// TIA Portal V16 export
// export: Created 2023-06-21T17:06:27.0231194Z, ExportSetting WithDefaults, DisplayName Totally Integrated Automation Portal, DisplayVersion V16 Update 4, DisplayName TIA Portal Version Control Interface, DisplayVersion V16 Update 2, DisplayName TIA Portal Openness, DisplayVersion V16 Update 4, DisplayName SINAMICS Startdrive Advanced, DisplayVersion V16, DisplayName SINAMICS Startdrive G130, G150, S120, S150, SINAMICS MV, S210, DisplayVersion V16, DisplayName SINAMICS Startdrive G110M, G120, G120C, G120D, G120P, DisplayVersion V16, DisplayName STEP 7 Professional, DisplayVersion V16 Update 4, DisplayName STEP 7 Safety, DisplayVersion V16, DisplayName Soft Starter ES, DisplayVersion V16, DisplayName WinCC Advanced, DisplayVersion V16 Update 4
FUNCTION "Data_Treatment" : Void   // FC2, LAD
{ S7_Optimized_Access := 'TRUE' }
VERSION : 0.1
// stored: AutoNumber true, IsIECCheckEnabled false, SetENOAutomatically false, UDAEnableTagReadback false
BEGIN

REGION Network 1: Extrusora 1
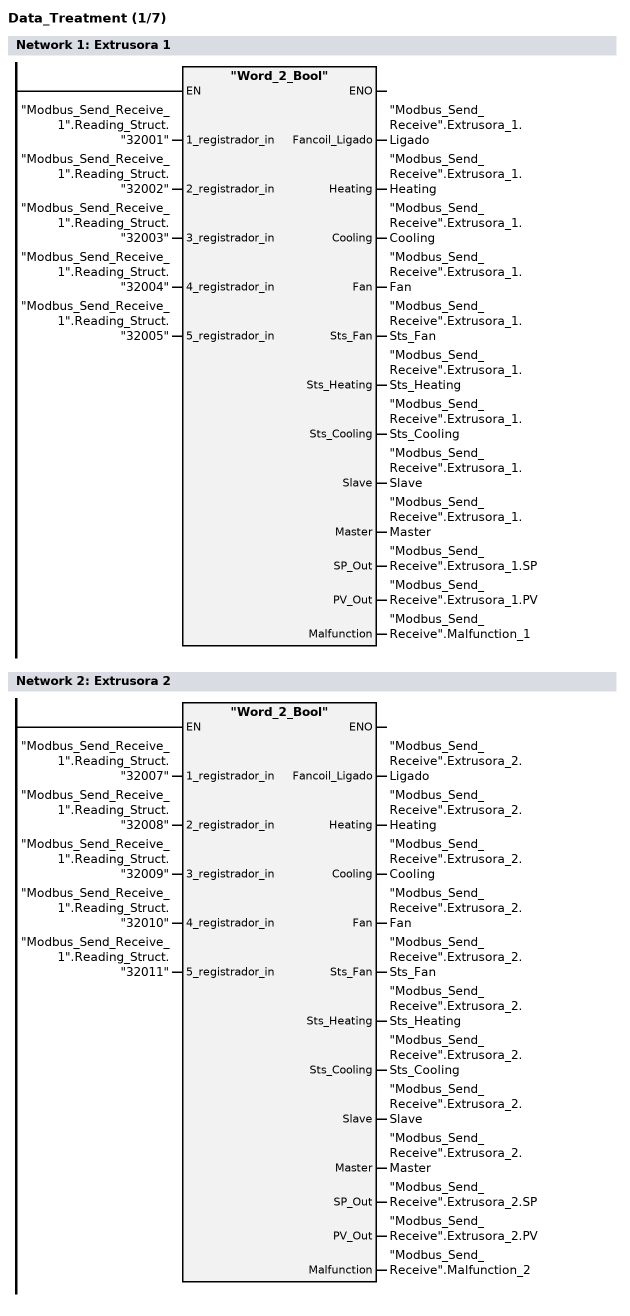
   RUNG wire#powerrail
      "Word_2_Bool"("1_registrador_in" := "Modbus_Send_Receive_1".Reading_Struct."32001", "2_registrador_in" := "Modbus_Send_Receive_1".Reading_Struct."32002", "3_registrador_in" := "Modbus_Send_Receive_1".Reading_Struct."32003", "4_registrador_in" := "Modbus_Send_Receive_1".Reading_Struct."32004", "5_registrador_in" := "Modbus_Send_Receive_1".Reading_Struct."32005", Fancoil_Ligado => "Modbus_Send_Receive".Extrusora_1.Ligado, Heating => "Modbus_Send_Receive".Extrusora_1.Heating, Cooling => "Modbus_Send_Receive".Extrusora_1.Cooling, Fan => "Modbus_Send_Receive".Extrusora_1.Fan, Sts_Fan => "Modbus_Send_Receive".Extrusora_1.Sts_Fan, Sts_Heating => "Modbus_Send_Receive".Extrusora_1.Sts_Heating, Sts_Cooling => "Modbus_Send_Receive".Extrusora_1.Sts_Cooling, Slave => "Modbus_Send_Receive".Extrusora_1.Slave, Master => "Modbus_Send_Receive".Extrusora_1.Master, SP_Out => "Modbus_Send_Receive".Extrusora_1.SP, PV_Out => "Modbus_Send_Receive".Extrusora_1.PV, Malfunction => "Modbus_Send_Receive".Malfunction_1)
   END_RUNG
   // the same network as SCL:
   "Word_2_Bool"("1_registrador_in" := "Modbus_Send_Receive_1".Reading_Struct."32001",
                 "2_registrador_in" := "Modbus_Send_Receive_1".Reading_Struct."32002",
                 "3_registrador_in" := "Modbus_Send_Receive_1".Reading_Struct."32003",
                 "4_registrador_in" := "Modbus_Send_Receive_1".Reading_Struct."32004",
                 "5_registrador_in" := "Modbus_Send_Receive_1".Reading_Struct."32005",
                 Fancoil_Ligado => "Modbus_Send_Receive".Extrusora_1.Ligado,
                 Heating => "Modbus_Send_Receive".Extrusora_1.Heating,
                 Cooling => "Modbus_Send_Receive".Extrusora_1.Cooling,
                 Fan => "Modbus_Send_Receive".Extrusora_1.Fan,
                 Sts_Fan => "Modbus_Send_Receive".Extrusora_1.Sts_Fan,
                 Sts_Heating => "Modbus_Send_Receive".Extrusora_1.Sts_Heating,
                 Sts_Cooling => "Modbus_Send_Receive".Extrusora_1.Sts_Cooling,
                 Slave => "Modbus_Send_Receive".Extrusora_1.Slave,
                 Master => "Modbus_Send_Receive".Extrusora_1.Master,
                 SP_Out => "Modbus_Send_Receive".Extrusora_1.SP,
                 PV_Out => "Modbus_Send_Receive".Extrusora_1.PV,
                 Malfunction => "Modbus_Send_Receive".Malfunction_1);
END_REGION

REGION Network 2: Extrusora 2
   RUNG wire#powerrail
      "Word_2_Bool"("1_registrador_in" := "Modbus_Send_Receive_1".Reading_Struct."32007", "2_registrador_in" := "Modbus_Send_Receive_1".Reading_Struct."32008", "3_registrador_in" := "Modbus_Send_Receive_1".Reading_Struct."32009", "4_registrador_in" := "Modbus_Send_Receive_1".Reading_Struct."32010", "5_registrador_in" := "Modbus_Send_Receive_1".Reading_Struct."32011", Fancoil_Ligado => "Modbus_Send_Receive".Extrusora_2.Ligado, Heating => "Modbus_Send_Receive".Extrusora_2.Heating, Cooling => "Modbus_Send_Receive".Extrusora_2.Cooling, Fan => "Modbus_Send_Receive".Extrusora_2.Fan, Sts_Fan => "Modbus_Send_Receive".Extrusora_2.Sts_Fan, Sts_Heating => "Modbus_Send_Receive".Extrusora_2.Sts_Heating, Sts_Cooling => "Modbus_Send_Receive".Extrusora_2.Sts_Cooling, Slave => "Modbus_Send_Receive".Extrusora_2.Slave, Master => "Modbus_Send_Receive".Extrusora_2.Master, SP_Out => "Modbus_Send_Receive".Extrusora_2.SP, PV_Out => "Modbus_Send_Receive".Extrusora_2.PV, Malfunction => "Modbus_Send_Receive".Malfunction_2)
   END_RUNG
   // the same network as SCL:
   "Word_2_Bool"("1_registrador_in" := "Modbus_Send_Receive_1".Reading_Struct."32007",
                 "2_registrador_in" := "Modbus_Send_Receive_1".Reading_Struct."32008",
                 "3_registrador_in" := "Modbus_Send_Receive_1".Reading_Struct."32009",
                 "4_registrador_in" := "Modbus_Send_Receive_1".Reading_Struct."32010",
                 "5_registrador_in" := "Modbus_Send_Receive_1".Reading_Struct."32011",
                 Fancoil_Ligado => "Modbus_Send_Receive".Extrusora_2.Ligado,
                 Heating => "Modbus_Send_Receive".Extrusora_2.Heating,
                 Cooling => "Modbus_Send_Receive".Extrusora_2.Cooling,
                 Fan => "Modbus_Send_Receive".Extrusora_2.Fan,
                 Sts_Fan => "Modbus_Send_Receive".Extrusora_2.Sts_Fan,
                 Sts_Heating => "Modbus_Send_Receive".Extrusora_2.Sts_Heating,
                 Sts_Cooling => "Modbus_Send_Receive".Extrusora_2.Sts_Cooling,
                 Slave => "Modbus_Send_Receive".Extrusora_2.Slave,
                 Master => "Modbus_Send_Receive".Extrusora_2.Master,
                 SP_Out => "Modbus_Send_Receive".Extrusora_2.SP,
                 PV_Out => "Modbus_Send_Receive".Extrusora_2.PV,
                 Malfunction => "Modbus_Send_Receive".Malfunction_2);
END_REGION

REGION Network 3: Extrusora 3
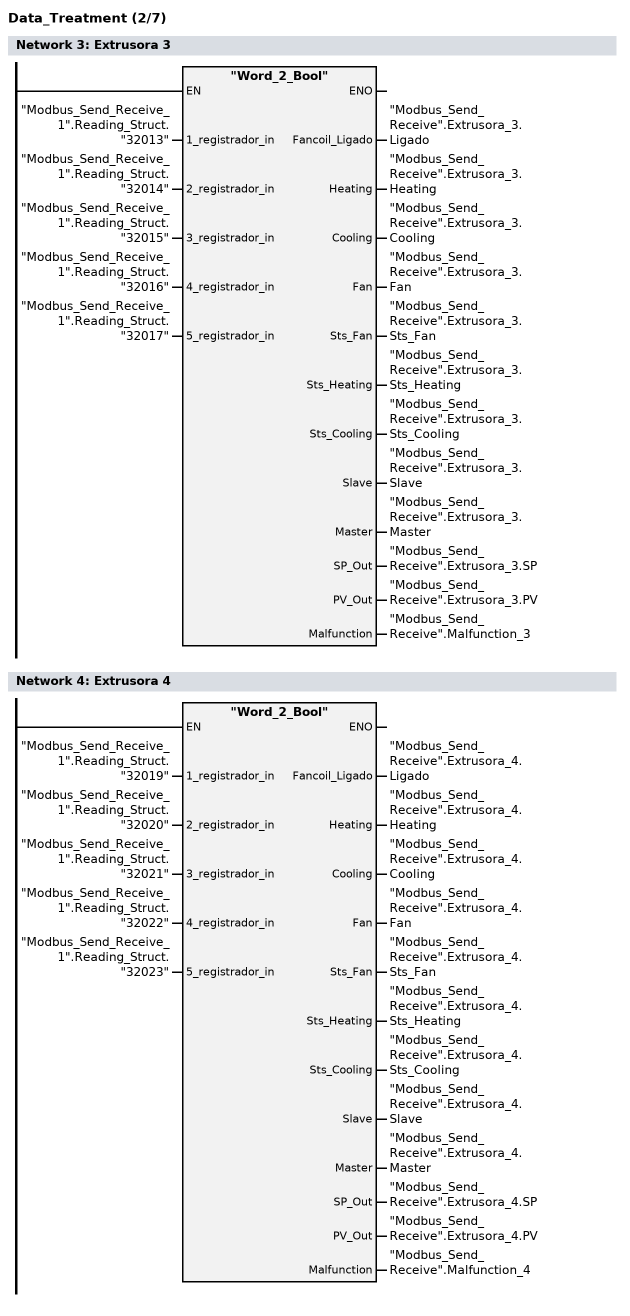
   RUNG wire#powerrail
      "Word_2_Bool"("1_registrador_in" := "Modbus_Send_Receive_1".Reading_Struct."32013", "2_registrador_in" := "Modbus_Send_Receive_1".Reading_Struct."32014", "3_registrador_in" := "Modbus_Send_Receive_1".Reading_Struct."32015", "4_registrador_in" := "Modbus_Send_Receive_1".Reading_Struct."32016", "5_registrador_in" := "Modbus_Send_Receive_1".Reading_Struct."32017", Fancoil_Ligado => "Modbus_Send_Receive".Extrusora_3.Ligado, Heating => "Modbus_Send_Receive".Extrusora_3.Heating, Cooling => "Modbus_Send_Receive".Extrusora_3.Cooling, Fan => "Modbus_Send_Receive".Extrusora_3.Fan, Sts_Fan => "Modbus_Send_Receive".Extrusora_3.Sts_Fan, Sts_Heating => "Modbus_Send_Receive".Extrusora_3.Sts_Heating, Sts_Cooling => "Modbus_Send_Receive".Extrusora_3.Sts_Cooling, Slave => "Modbus_Send_Receive".Extrusora_3.Slave, Master => "Modbus_Send_Receive".Extrusora_3.Master, SP_Out => "Modbus_Send_Receive".Extrusora_3.SP, PV_Out => "Modbus_Send_Receive".Extrusora_3.PV, Malfunction => "Modbus_Send_Receive".Malfunction_3)
   END_RUNG
   // the same network as SCL:
   "Word_2_Bool"("1_registrador_in" := "Modbus_Send_Receive_1".Reading_Struct."32013",
                 "2_registrador_in" := "Modbus_Send_Receive_1".Reading_Struct."32014",
                 "3_registrador_in" := "Modbus_Send_Receive_1".Reading_Struct."32015",
                 "4_registrador_in" := "Modbus_Send_Receive_1".Reading_Struct."32016",
                 "5_registrador_in" := "Modbus_Send_Receive_1".Reading_Struct."32017",
                 Fancoil_Ligado => "Modbus_Send_Receive".Extrusora_3.Ligado,
                 Heating => "Modbus_Send_Receive".Extrusora_3.Heating,
                 Cooling => "Modbus_Send_Receive".Extrusora_3.Cooling,
                 Fan => "Modbus_Send_Receive".Extrusora_3.Fan,
                 Sts_Fan => "Modbus_Send_Receive".Extrusora_3.Sts_Fan,
                 Sts_Heating => "Modbus_Send_Receive".Extrusora_3.Sts_Heating,
                 Sts_Cooling => "Modbus_Send_Receive".Extrusora_3.Sts_Cooling,
                 Slave => "Modbus_Send_Receive".Extrusora_3.Slave,
                 Master => "Modbus_Send_Receive".Extrusora_3.Master,
                 SP_Out => "Modbus_Send_Receive".Extrusora_3.SP,
                 PV_Out => "Modbus_Send_Receive".Extrusora_3.PV,
                 Malfunction => "Modbus_Send_Receive".Malfunction_3);
END_REGION

REGION Network 4: Extrusora 4
   RUNG wire#powerrail
      "Word_2_Bool"("1_registrador_in" := "Modbus_Send_Receive_1".Reading_Struct."32019", "2_registrador_in" := "Modbus_Send_Receive_1".Reading_Struct."32020", "3_registrador_in" := "Modbus_Send_Receive_1".Reading_Struct."32021", "4_registrador_in" := "Modbus_Send_Receive_1".Reading_Struct."32022", "5_registrador_in" := "Modbus_Send_Receive_1".Reading_Struct."32023", Fancoil_Ligado => "Modbus_Send_Receive".Extrusora_4.Ligado, Heating => "Modbus_Send_Receive".Extrusora_4.Heating, Cooling => "Modbus_Send_Receive".Extrusora_4.Cooling, Fan => "Modbus_Send_Receive".Extrusora_4.Fan, Sts_Fan => "Modbus_Send_Receive".Extrusora_4.Sts_Fan, Sts_Heating => "Modbus_Send_Receive".Extrusora_4.Sts_Heating, Sts_Cooling => "Modbus_Send_Receive".Extrusora_4.Sts_Cooling, Slave => "Modbus_Send_Receive".Extrusora_4.Slave, Master => "Modbus_Send_Receive".Extrusora_4.Master, SP_Out => "Modbus_Send_Receive".Extrusora_4.SP, PV_Out => "Modbus_Send_Receive".Extrusora_4.PV, Malfunction => "Modbus_Send_Receive".Malfunction_4)
   END_RUNG
   // the same network as SCL:
   "Word_2_Bool"("1_registrador_in" := "Modbus_Send_Receive_1".Reading_Struct."32019",
                 "2_registrador_in" := "Modbus_Send_Receive_1".Reading_Struct."32020",
                 "3_registrador_in" := "Modbus_Send_Receive_1".Reading_Struct."32021",
                 "4_registrador_in" := "Modbus_Send_Receive_1".Reading_Struct."32022",
                 "5_registrador_in" := "Modbus_Send_Receive_1".Reading_Struct."32023",
                 Fancoil_Ligado => "Modbus_Send_Receive".Extrusora_4.Ligado,
                 Heating => "Modbus_Send_Receive".Extrusora_4.Heating,
                 Cooling => "Modbus_Send_Receive".Extrusora_4.Cooling,
                 Fan => "Modbus_Send_Receive".Extrusora_4.Fan,
                 Sts_Fan => "Modbus_Send_Receive".Extrusora_4.Sts_Fan,
                 Sts_Heating => "Modbus_Send_Receive".Extrusora_4.Sts_Heating,
                 Sts_Cooling => "Modbus_Send_Receive".Extrusora_4.Sts_Cooling,
                 Slave => "Modbus_Send_Receive".Extrusora_4.Slave,
                 Master => "Modbus_Send_Receive".Extrusora_4.Master,
                 SP_Out => "Modbus_Send_Receive".Extrusora_4.SP,
                 PV_Out => "Modbus_Send_Receive".Extrusora_4.PV,
                 Malfunction => "Modbus_Send_Receive".Malfunction_4);
END_REGION

REGION Network 5: Extrusora 5
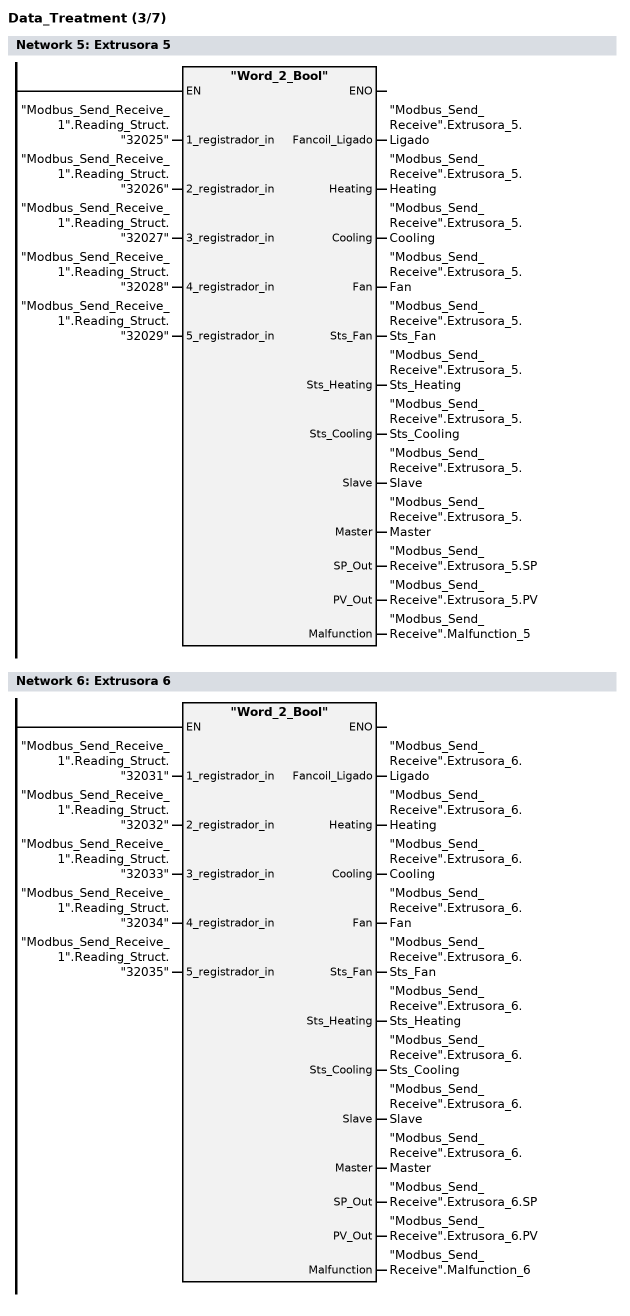
   RUNG wire#powerrail
      "Word_2_Bool"("1_registrador_in" := "Modbus_Send_Receive_1".Reading_Struct."32025", "2_registrador_in" := "Modbus_Send_Receive_1".Reading_Struct."32026", "3_registrador_in" := "Modbus_Send_Receive_1".Reading_Struct."32027", "4_registrador_in" := "Modbus_Send_Receive_1".Reading_Struct."32028", "5_registrador_in" := "Modbus_Send_Receive_1".Reading_Struct."32029", Fancoil_Ligado => "Modbus_Send_Receive".Extrusora_5.Ligado, Heating => "Modbus_Send_Receive".Extrusora_5.Heating, Cooling => "Modbus_Send_Receive".Extrusora_5.Cooling, Fan => "Modbus_Send_Receive".Extrusora_5.Fan, Sts_Fan => "Modbus_Send_Receive".Extrusora_5.Sts_Fan, Sts_Heating => "Modbus_Send_Receive".Extrusora_5.Sts_Heating, Sts_Cooling => "Modbus_Send_Receive".Extrusora_5.Sts_Cooling, Slave => "Modbus_Send_Receive".Extrusora_5.Slave, Master => "Modbus_Send_Receive".Extrusora_5.Master, SP_Out => "Modbus_Send_Receive".Extrusora_5.SP, PV_Out => "Modbus_Send_Receive".Extrusora_5.PV, Malfunction => "Modbus_Send_Receive".Malfunction_5)
   END_RUNG
   // the same network as SCL:
   "Word_2_Bool"("1_registrador_in" := "Modbus_Send_Receive_1".Reading_Struct."32025",
                 "2_registrador_in" := "Modbus_Send_Receive_1".Reading_Struct."32026",
                 "3_registrador_in" := "Modbus_Send_Receive_1".Reading_Struct."32027",
                 "4_registrador_in" := "Modbus_Send_Receive_1".Reading_Struct."32028",
                 "5_registrador_in" := "Modbus_Send_Receive_1".Reading_Struct."32029",
                 Fancoil_Ligado => "Modbus_Send_Receive".Extrusora_5.Ligado,
                 Heating => "Modbus_Send_Receive".Extrusora_5.Heating,
                 Cooling => "Modbus_Send_Receive".Extrusora_5.Cooling,
                 Fan => "Modbus_Send_Receive".Extrusora_5.Fan,
                 Sts_Fan => "Modbus_Send_Receive".Extrusora_5.Sts_Fan,
                 Sts_Heating => "Modbus_Send_Receive".Extrusora_5.Sts_Heating,
                 Sts_Cooling => "Modbus_Send_Receive".Extrusora_5.Sts_Cooling,
                 Slave => "Modbus_Send_Receive".Extrusora_5.Slave,
                 Master => "Modbus_Send_Receive".Extrusora_5.Master,
                 SP_Out => "Modbus_Send_Receive".Extrusora_5.SP,
                 PV_Out => "Modbus_Send_Receive".Extrusora_5.PV,
                 Malfunction => "Modbus_Send_Receive".Malfunction_5);
END_REGION

REGION Network 6: Extrusora 6
   RUNG wire#powerrail
      "Word_2_Bool"("1_registrador_in" := "Modbus_Send_Receive_1".Reading_Struct."32031", "2_registrador_in" := "Modbus_Send_Receive_1".Reading_Struct."32032", "3_registrador_in" := "Modbus_Send_Receive_1".Reading_Struct."32033", "4_registrador_in" := "Modbus_Send_Receive_1".Reading_Struct."32034", "5_registrador_in" := "Modbus_Send_Receive_1".Reading_Struct."32035", Fancoil_Ligado => "Modbus_Send_Receive".Extrusora_6.Ligado, Heating => "Modbus_Send_Receive".Extrusora_6.Heating, Cooling => "Modbus_Send_Receive".Extrusora_6.Cooling, Fan => "Modbus_Send_Receive".Extrusora_6.Fan, Sts_Fan => "Modbus_Send_Receive".Extrusora_6.Sts_Fan, Sts_Heating => "Modbus_Send_Receive".Extrusora_6.Sts_Heating, Sts_Cooling => "Modbus_Send_Receive".Extrusora_6.Sts_Cooling, Slave => "Modbus_Send_Receive".Extrusora_6.Slave, Master => "Modbus_Send_Receive".Extrusora_6.Master, SP_Out => "Modbus_Send_Receive".Extrusora_6.SP, PV_Out => "Modbus_Send_Receive".Extrusora_6.PV, Malfunction => "Modbus_Send_Receive".Malfunction_6)
   END_RUNG
   // the same network as SCL:
   "Word_2_Bool"("1_registrador_in" := "Modbus_Send_Receive_1".Reading_Struct."32031",
                 "2_registrador_in" := "Modbus_Send_Receive_1".Reading_Struct."32032",
                 "3_registrador_in" := "Modbus_Send_Receive_1".Reading_Struct."32033",
                 "4_registrador_in" := "Modbus_Send_Receive_1".Reading_Struct."32034",
                 "5_registrador_in" := "Modbus_Send_Receive_1".Reading_Struct."32035",
                 Fancoil_Ligado => "Modbus_Send_Receive".Extrusora_6.Ligado,
                 Heating => "Modbus_Send_Receive".Extrusora_6.Heating,
                 Cooling => "Modbus_Send_Receive".Extrusora_6.Cooling,
                 Fan => "Modbus_Send_Receive".Extrusora_6.Fan,
                 Sts_Fan => "Modbus_Send_Receive".Extrusora_6.Sts_Fan,
                 Sts_Heating => "Modbus_Send_Receive".Extrusora_6.Sts_Heating,
                 Sts_Cooling => "Modbus_Send_Receive".Extrusora_6.Sts_Cooling,
                 Slave => "Modbus_Send_Receive".Extrusora_6.Slave,
                 Master => "Modbus_Send_Receive".Extrusora_6.Master,
                 SP_Out => "Modbus_Send_Receive".Extrusora_6.SP,
                 PV_Out => "Modbus_Send_Receive".Extrusora_6.PV,
                 Malfunction => "Modbus_Send_Receive".Malfunction_6);
END_REGION

REGION Network 7: Extrusora 8
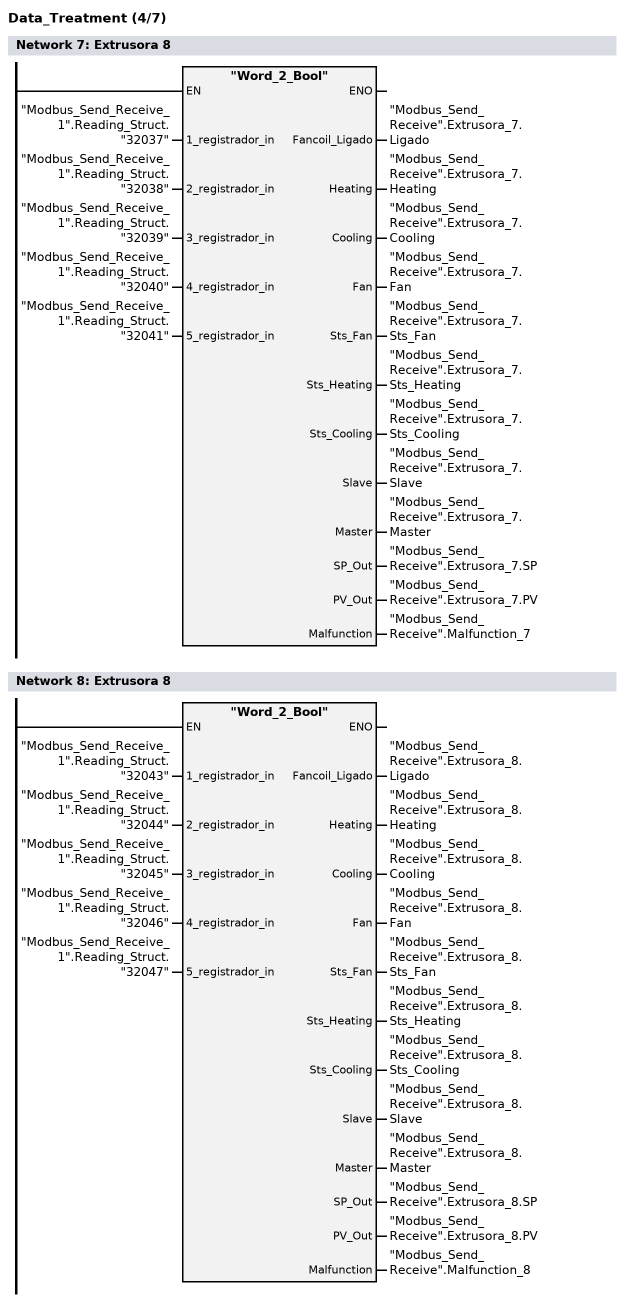
   RUNG wire#powerrail
      "Word_2_Bool"("1_registrador_in" := "Modbus_Send_Receive_1".Reading_Struct."32037", "2_registrador_in" := "Modbus_Send_Receive_1".Reading_Struct."32038", "3_registrador_in" := "Modbus_Send_Receive_1".Reading_Struct."32039", "4_registrador_in" := "Modbus_Send_Receive_1".Reading_Struct."32040", "5_registrador_in" := "Modbus_Send_Receive_1".Reading_Struct."32041", Fancoil_Ligado => "Modbus_Send_Receive".Extrusora_7.Ligado, Heating => "Modbus_Send_Receive".Extrusora_7.Heating, Cooling => "Modbus_Send_Receive".Extrusora_7.Cooling, Fan => "Modbus_Send_Receive".Extrusora_7.Fan, Sts_Fan => "Modbus_Send_Receive".Extrusora_7.Sts_Fan, Sts_Heating => "Modbus_Send_Receive".Extrusora_7.Sts_Heating, Sts_Cooling => "Modbus_Send_Receive".Extrusora_7.Sts_Cooling, Slave => "Modbus_Send_Receive".Extrusora_7.Slave, Master => "Modbus_Send_Receive".Extrusora_7.Master, SP_Out => "Modbus_Send_Receive".Extrusora_7.SP, PV_Out => "Modbus_Send_Receive".Extrusora_7.PV, Malfunction => "Modbus_Send_Receive".Malfunction_7)
   END_RUNG
   // the same network as SCL:
   "Word_2_Bool"("1_registrador_in" := "Modbus_Send_Receive_1".Reading_Struct."32037",
                 "2_registrador_in" := "Modbus_Send_Receive_1".Reading_Struct."32038",
                 "3_registrador_in" := "Modbus_Send_Receive_1".Reading_Struct."32039",
                 "4_registrador_in" := "Modbus_Send_Receive_1".Reading_Struct."32040",
                 "5_registrador_in" := "Modbus_Send_Receive_1".Reading_Struct."32041",
                 Fancoil_Ligado => "Modbus_Send_Receive".Extrusora_7.Ligado,
                 Heating => "Modbus_Send_Receive".Extrusora_7.Heating,
                 Cooling => "Modbus_Send_Receive".Extrusora_7.Cooling,
                 Fan => "Modbus_Send_Receive".Extrusora_7.Fan,
                 Sts_Fan => "Modbus_Send_Receive".Extrusora_7.Sts_Fan,
                 Sts_Heating => "Modbus_Send_Receive".Extrusora_7.Sts_Heating,
                 Sts_Cooling => "Modbus_Send_Receive".Extrusora_7.Sts_Cooling,
                 Slave => "Modbus_Send_Receive".Extrusora_7.Slave,
                 Master => "Modbus_Send_Receive".Extrusora_7.Master,
                 SP_Out => "Modbus_Send_Receive".Extrusora_7.SP,
                 PV_Out => "Modbus_Send_Receive".Extrusora_7.PV,
                 Malfunction => "Modbus_Send_Receive".Malfunction_7);
END_REGION

REGION Network 8: Extrusora 8
   RUNG wire#powerrail
      "Word_2_Bool"("1_registrador_in" := "Modbus_Send_Receive_1".Reading_Struct."32043", "2_registrador_in" := "Modbus_Send_Receive_1".Reading_Struct."32044", "3_registrador_in" := "Modbus_Send_Receive_1".Reading_Struct."32045", "4_registrador_in" := "Modbus_Send_Receive_1".Reading_Struct."32046", "5_registrador_in" := "Modbus_Send_Receive_1".Reading_Struct."32047", Fancoil_Ligado => "Modbus_Send_Receive".Extrusora_8.Ligado, Heating => "Modbus_Send_Receive".Extrusora_8.Heating, Cooling => "Modbus_Send_Receive".Extrusora_8.Cooling, Fan => "Modbus_Send_Receive".Extrusora_8.Fan, Sts_Fan => "Modbus_Send_Receive".Extrusora_8.Sts_Fan, Sts_Heating => "Modbus_Send_Receive".Extrusora_8.Sts_Heating, Sts_Cooling => "Modbus_Send_Receive".Extrusora_8.Sts_Cooling, Slave => "Modbus_Send_Receive".Extrusora_8.Slave, Master => "Modbus_Send_Receive".Extrusora_8.Master, SP_Out => "Modbus_Send_Receive".Extrusora_8.SP, PV_Out => "Modbus_Send_Receive".Extrusora_8.PV, Malfunction => "Modbus_Send_Receive".Malfunction_8)
   END_RUNG
   // the same network as SCL:
   "Word_2_Bool"("1_registrador_in" := "Modbus_Send_Receive_1".Reading_Struct."32043",
                 "2_registrador_in" := "Modbus_Send_Receive_1".Reading_Struct."32044",
                 "3_registrador_in" := "Modbus_Send_Receive_1".Reading_Struct."32045",
                 "4_registrador_in" := "Modbus_Send_Receive_1".Reading_Struct."32046",
                 "5_registrador_in" := "Modbus_Send_Receive_1".Reading_Struct."32047",
                 Fancoil_Ligado => "Modbus_Send_Receive".Extrusora_8.Ligado,
                 Heating => "Modbus_Send_Receive".Extrusora_8.Heating,
                 Cooling => "Modbus_Send_Receive".Extrusora_8.Cooling,
                 Fan => "Modbus_Send_Receive".Extrusora_8.Fan,
                 Sts_Fan => "Modbus_Send_Receive".Extrusora_8.Sts_Fan,
                 Sts_Heating => "Modbus_Send_Receive".Extrusora_8.Sts_Heating,
                 Sts_Cooling => "Modbus_Send_Receive".Extrusora_8.Sts_Cooling,
                 Slave => "Modbus_Send_Receive".Extrusora_8.Slave,
                 Master => "Modbus_Send_Receive".Extrusora_8.Master,
                 SP_Out => "Modbus_Send_Receive".Extrusora_8.SP,
                 PV_Out => "Modbus_Send_Receive".Extrusora_8.PV,
                 Malfunction => "Modbus_Send_Receive".Malfunction_8);
END_REGION

REGION Network 9: Extrusora 9
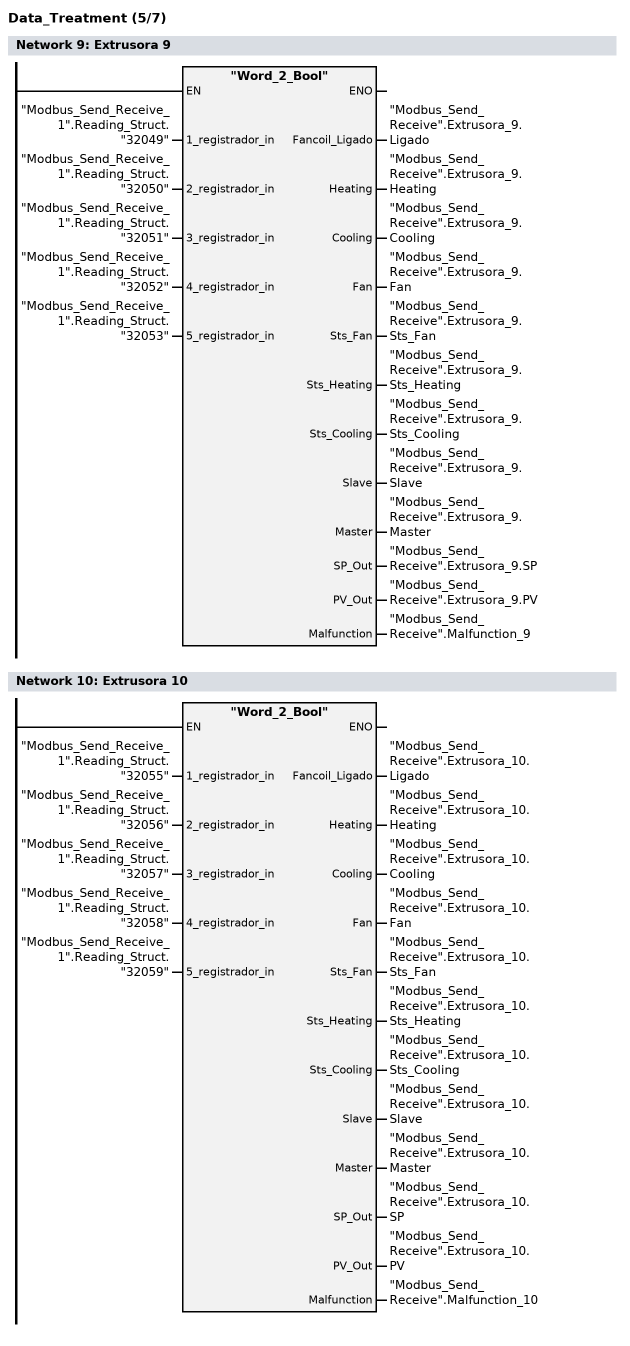
   RUNG wire#powerrail
      "Word_2_Bool"("1_registrador_in" := "Modbus_Send_Receive_1".Reading_Struct."32049", "2_registrador_in" := "Modbus_Send_Receive_1".Reading_Struct."32050", "3_registrador_in" := "Modbus_Send_Receive_1".Reading_Struct."32051", "4_registrador_in" := "Modbus_Send_Receive_1".Reading_Struct."32052", "5_registrador_in" := "Modbus_Send_Receive_1".Reading_Struct."32053", Fancoil_Ligado => "Modbus_Send_Receive".Extrusora_9.Ligado, Heating => "Modbus_Send_Receive".Extrusora_9.Heating, Cooling => "Modbus_Send_Receive".Extrusora_9.Cooling, Fan => "Modbus_Send_Receive".Extrusora_9.Fan, Sts_Fan => "Modbus_Send_Receive".Extrusora_9.Sts_Fan, Sts_Heating => "Modbus_Send_Receive".Extrusora_9.Sts_Heating, Sts_Cooling => "Modbus_Send_Receive".Extrusora_9.Sts_Cooling, Slave => "Modbus_Send_Receive".Extrusora_9.Slave, Master => "Modbus_Send_Receive".Extrusora_9.Master, SP_Out => "Modbus_Send_Receive".Extrusora_9.SP, PV_Out => "Modbus_Send_Receive".Extrusora_9.PV, Malfunction => "Modbus_Send_Receive".Malfunction_9)
   END_RUNG
   // the same network as SCL:
   "Word_2_Bool"("1_registrador_in" := "Modbus_Send_Receive_1".Reading_Struct."32049",
                 "2_registrador_in" := "Modbus_Send_Receive_1".Reading_Struct."32050",
                 "3_registrador_in" := "Modbus_Send_Receive_1".Reading_Struct."32051",
                 "4_registrador_in" := "Modbus_Send_Receive_1".Reading_Struct."32052",
                 "5_registrador_in" := "Modbus_Send_Receive_1".Reading_Struct."32053",
                 Fancoil_Ligado => "Modbus_Send_Receive".Extrusora_9.Ligado,
                 Heating => "Modbus_Send_Receive".Extrusora_9.Heating,
                 Cooling => "Modbus_Send_Receive".Extrusora_9.Cooling,
                 Fan => "Modbus_Send_Receive".Extrusora_9.Fan,
                 Sts_Fan => "Modbus_Send_Receive".Extrusora_9.Sts_Fan,
                 Sts_Heating => "Modbus_Send_Receive".Extrusora_9.Sts_Heating,
                 Sts_Cooling => "Modbus_Send_Receive".Extrusora_9.Sts_Cooling,
                 Slave => "Modbus_Send_Receive".Extrusora_9.Slave,
                 Master => "Modbus_Send_Receive".Extrusora_9.Master,
                 SP_Out => "Modbus_Send_Receive".Extrusora_9.SP,
                 PV_Out => "Modbus_Send_Receive".Extrusora_9.PV,
                 Malfunction => "Modbus_Send_Receive".Malfunction_9);
END_REGION

REGION Network 10: Extrusora 10
   RUNG wire#powerrail
      "Word_2_Bool"("1_registrador_in" := "Modbus_Send_Receive_1".Reading_Struct."32055", "2_registrador_in" := "Modbus_Send_Receive_1".Reading_Struct."32056", "3_registrador_in" := "Modbus_Send_Receive_1".Reading_Struct."32057", "4_registrador_in" := "Modbus_Send_Receive_1".Reading_Struct."32058", "5_registrador_in" := "Modbus_Send_Receive_1".Reading_Struct."32059", Fancoil_Ligado => "Modbus_Send_Receive".Extrusora_10.Ligado, Heating => "Modbus_Send_Receive".Extrusora_10.Heating, Cooling => "Modbus_Send_Receive".Extrusora_10.Cooling, Fan => "Modbus_Send_Receive".Extrusora_10.Fan, Sts_Fan => "Modbus_Send_Receive".Extrusora_10.Sts_Fan, Sts_Heating => "Modbus_Send_Receive".Extrusora_10.Sts_Heating, Sts_Cooling => "Modbus_Send_Receive".Extrusora_10.Sts_Cooling, Slave => "Modbus_Send_Receive".Extrusora_10.Slave, Master => "Modbus_Send_Receive".Extrusora_10.Master, SP_Out => "Modbus_Send_Receive".Extrusora_10.SP, PV_Out => "Modbus_Send_Receive".Extrusora_10.PV, Malfunction => "Modbus_Send_Receive".Malfunction_10)
   END_RUNG
   // the same network as SCL:
   "Word_2_Bool"("1_registrador_in" := "Modbus_Send_Receive_1".Reading_Struct."32055",
                 "2_registrador_in" := "Modbus_Send_Receive_1".Reading_Struct."32056",
                 "3_registrador_in" := "Modbus_Send_Receive_1".Reading_Struct."32057",
                 "4_registrador_in" := "Modbus_Send_Receive_1".Reading_Struct."32058",
                 "5_registrador_in" := "Modbus_Send_Receive_1".Reading_Struct."32059",
                 Fancoil_Ligado => "Modbus_Send_Receive".Extrusora_10.Ligado,
                 Heating => "Modbus_Send_Receive".Extrusora_10.Heating,
                 Cooling => "Modbus_Send_Receive".Extrusora_10.Cooling,
                 Fan => "Modbus_Send_Receive".Extrusora_10.Fan,
                 Sts_Fan => "Modbus_Send_Receive".Extrusora_10.Sts_Fan,
                 Sts_Heating => "Modbus_Send_Receive".Extrusora_10.Sts_Heating,
                 Sts_Cooling => "Modbus_Send_Receive".Extrusora_10.Sts_Cooling,
                 Slave => "Modbus_Send_Receive".Extrusora_10.Slave,
                 Master => "Modbus_Send_Receive".Extrusora_10.Master,
                 SP_Out => "Modbus_Send_Receive".Extrusora_10.SP,
                 PV_Out => "Modbus_Send_Receive".Extrusora_10.PV,
                 Malfunction => "Modbus_Send_Receive".Malfunction_10);
END_REGION

REGION Network 11: Extrusora 11
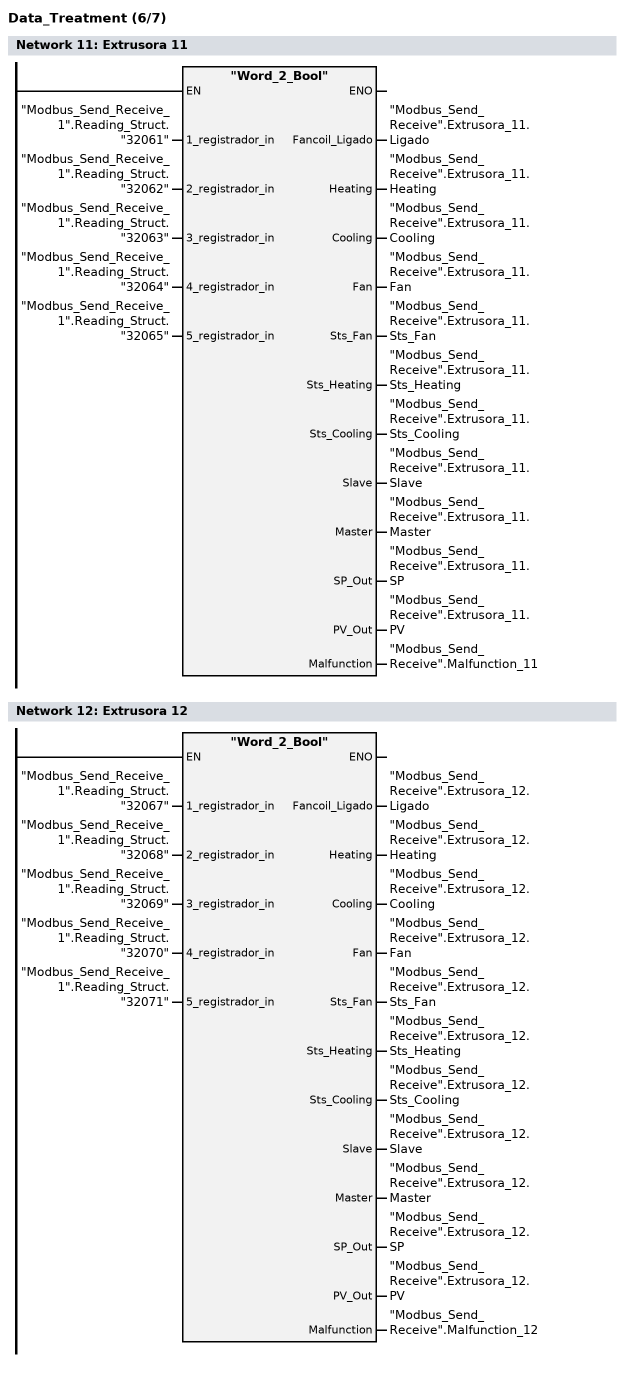
   RUNG wire#powerrail
      "Word_2_Bool"("1_registrador_in" := "Modbus_Send_Receive_1".Reading_Struct."32061", "2_registrador_in" := "Modbus_Send_Receive_1".Reading_Struct."32062", "3_registrador_in" := "Modbus_Send_Receive_1".Reading_Struct."32063", "4_registrador_in" := "Modbus_Send_Receive_1".Reading_Struct."32064", "5_registrador_in" := "Modbus_Send_Receive_1".Reading_Struct."32065", Fancoil_Ligado => "Modbus_Send_Receive".Extrusora_11.Ligado, Heating => "Modbus_Send_Receive".Extrusora_11.Heating, Cooling => "Modbus_Send_Receive".Extrusora_11.Cooling, Fan => "Modbus_Send_Receive".Extrusora_11.Fan, Sts_Fan => "Modbus_Send_Receive".Extrusora_11.Sts_Fan, Sts_Heating => "Modbus_Send_Receive".Extrusora_11.Sts_Heating, Sts_Cooling => "Modbus_Send_Receive".Extrusora_11.Sts_Cooling, Slave => "Modbus_Send_Receive".Extrusora_11.Slave, Master => "Modbus_Send_Receive".Extrusora_11.Master, SP_Out => "Modbus_Send_Receive".Extrusora_11.SP, PV_Out => "Modbus_Send_Receive".Extrusora_11.PV, Malfunction => "Modbus_Send_Receive".Malfunction_11)
   END_RUNG
   // the same network as SCL:
   "Word_2_Bool"("1_registrador_in" := "Modbus_Send_Receive_1".Reading_Struct."32061",
                 "2_registrador_in" := "Modbus_Send_Receive_1".Reading_Struct."32062",
                 "3_registrador_in" := "Modbus_Send_Receive_1".Reading_Struct."32063",
                 "4_registrador_in" := "Modbus_Send_Receive_1".Reading_Struct."32064",
                 "5_registrador_in" := "Modbus_Send_Receive_1".Reading_Struct."32065",
                 Fancoil_Ligado => "Modbus_Send_Receive".Extrusora_11.Ligado,
                 Heating => "Modbus_Send_Receive".Extrusora_11.Heating,
                 Cooling => "Modbus_Send_Receive".Extrusora_11.Cooling,
                 Fan => "Modbus_Send_Receive".Extrusora_11.Fan,
                 Sts_Fan => "Modbus_Send_Receive".Extrusora_11.Sts_Fan,
                 Sts_Heating => "Modbus_Send_Receive".Extrusora_11.Sts_Heating,
                 Sts_Cooling => "Modbus_Send_Receive".Extrusora_11.Sts_Cooling,
                 Slave => "Modbus_Send_Receive".Extrusora_11.Slave,
                 Master => "Modbus_Send_Receive".Extrusora_11.Master,
                 SP_Out => "Modbus_Send_Receive".Extrusora_11.SP,
                 PV_Out => "Modbus_Send_Receive".Extrusora_11.PV,
                 Malfunction => "Modbus_Send_Receive".Malfunction_11);
END_REGION

REGION Network 12: Extrusora 12
   RUNG wire#powerrail
      "Word_2_Bool"("1_registrador_in" := "Modbus_Send_Receive_1".Reading_Struct."32067", "2_registrador_in" := "Modbus_Send_Receive_1".Reading_Struct."32068", "3_registrador_in" := "Modbus_Send_Receive_1".Reading_Struct."32069", "4_registrador_in" := "Modbus_Send_Receive_1".Reading_Struct."32070", "5_registrador_in" := "Modbus_Send_Receive_1".Reading_Struct."32071", Fancoil_Ligado => "Modbus_Send_Receive".Extrusora_12.Ligado, Heating => "Modbus_Send_Receive".Extrusora_12.Heating, Cooling => "Modbus_Send_Receive".Extrusora_12.Cooling, Fan => "Modbus_Send_Receive".Extrusora_12.Fan, Sts_Fan => "Modbus_Send_Receive".Extrusora_12.Sts_Fan, Sts_Heating => "Modbus_Send_Receive".Extrusora_12.Sts_Heating, Sts_Cooling => "Modbus_Send_Receive".Extrusora_12.Sts_Cooling, Slave => "Modbus_Send_Receive".Extrusora_12.Slave, Master => "Modbus_Send_Receive".Extrusora_12.Master, SP_Out => "Modbus_Send_Receive".Extrusora_12.SP, PV_Out => "Modbus_Send_Receive".Extrusora_12.PV, Malfunction => "Modbus_Send_Receive".Malfunction_12)
   END_RUNG
   // the same network as SCL:
   "Word_2_Bool"("1_registrador_in" := "Modbus_Send_Receive_1".Reading_Struct."32067",
                 "2_registrador_in" := "Modbus_Send_Receive_1".Reading_Struct."32068",
                 "3_registrador_in" := "Modbus_Send_Receive_1".Reading_Struct."32069",
                 "4_registrador_in" := "Modbus_Send_Receive_1".Reading_Struct."32070",
                 "5_registrador_in" := "Modbus_Send_Receive_1".Reading_Struct."32071",
                 Fancoil_Ligado => "Modbus_Send_Receive".Extrusora_12.Ligado,
                 Heating => "Modbus_Send_Receive".Extrusora_12.Heating,
                 Cooling => "Modbus_Send_Receive".Extrusora_12.Cooling,
                 Fan => "Modbus_Send_Receive".Extrusora_12.Fan,
                 Sts_Fan => "Modbus_Send_Receive".Extrusora_12.Sts_Fan,
                 Sts_Heating => "Modbus_Send_Receive".Extrusora_12.Sts_Heating,
                 Sts_Cooling => "Modbus_Send_Receive".Extrusora_12.Sts_Cooling,
                 Slave => "Modbus_Send_Receive".Extrusora_12.Slave,
                 Master => "Modbus_Send_Receive".Extrusora_12.Master,
                 SP_Out => "Modbus_Send_Receive".Extrusora_12.SP,
                 PV_Out => "Modbus_Send_Receive".Extrusora_12.PV,
                 Malfunction => "Modbus_Send_Receive".Malfunction_12);
END_REGION

REGION Network 13: Extrusora 13
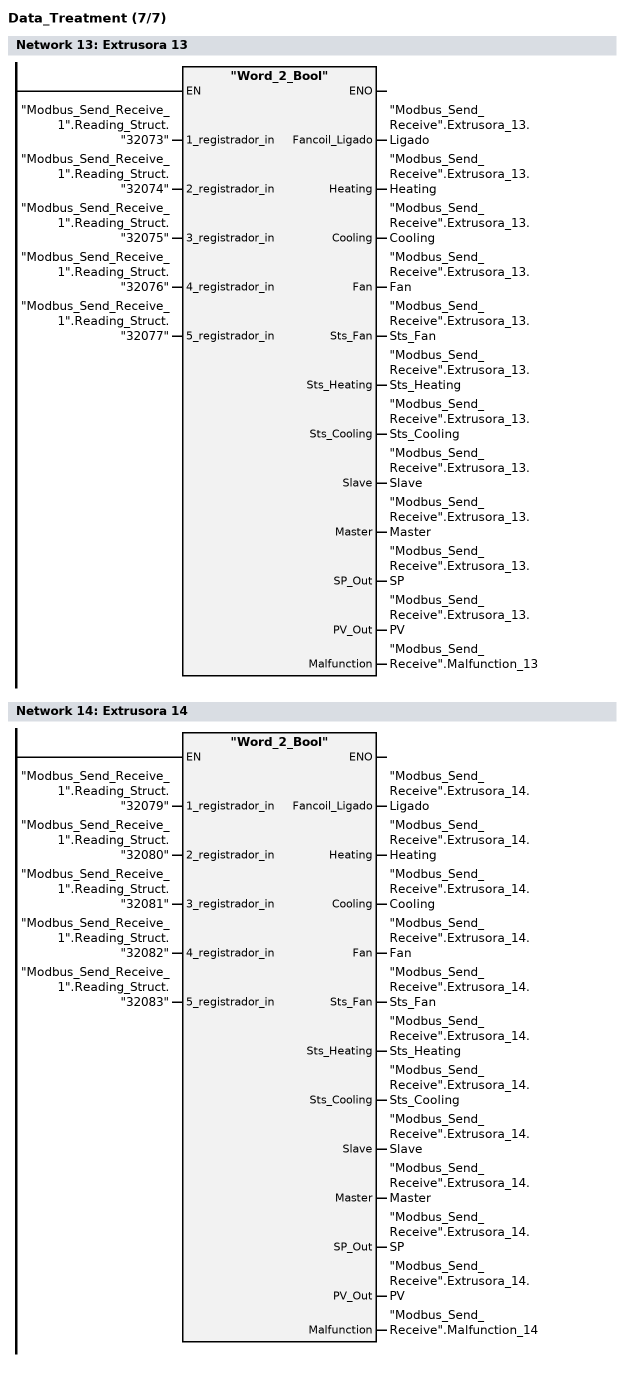
   RUNG wire#powerrail
      "Word_2_Bool"("1_registrador_in" := "Modbus_Send_Receive_1".Reading_Struct."32073", "2_registrador_in" := "Modbus_Send_Receive_1".Reading_Struct."32074", "3_registrador_in" := "Modbus_Send_Receive_1".Reading_Struct."32075", "4_registrador_in" := "Modbus_Send_Receive_1".Reading_Struct."32076", "5_registrador_in" := "Modbus_Send_Receive_1".Reading_Struct."32077", Fancoil_Ligado => "Modbus_Send_Receive".Extrusora_13.Ligado, Heating => "Modbus_Send_Receive".Extrusora_13.Heating, Cooling => "Modbus_Send_Receive".Extrusora_13.Cooling, Fan => "Modbus_Send_Receive".Extrusora_13.Fan, Sts_Fan => "Modbus_Send_Receive".Extrusora_13.Sts_Fan, Sts_Heating => "Modbus_Send_Receive".Extrusora_13.Sts_Heating, Sts_Cooling => "Modbus_Send_Receive".Extrusora_13.Sts_Cooling, Slave => "Modbus_Send_Receive".Extrusora_13.Slave, Master => "Modbus_Send_Receive".Extrusora_13.Master, SP_Out => "Modbus_Send_Receive".Extrusora_13.SP, PV_Out => "Modbus_Send_Receive".Extrusora_13.PV, Malfunction => "Modbus_Send_Receive".Malfunction_13)
   END_RUNG
   // the same network as SCL:
   "Word_2_Bool"("1_registrador_in" := "Modbus_Send_Receive_1".Reading_Struct."32073",
                 "2_registrador_in" := "Modbus_Send_Receive_1".Reading_Struct."32074",
                 "3_registrador_in" := "Modbus_Send_Receive_1".Reading_Struct."32075",
                 "4_registrador_in" := "Modbus_Send_Receive_1".Reading_Struct."32076",
                 "5_registrador_in" := "Modbus_Send_Receive_1".Reading_Struct."32077",
                 Fancoil_Ligado => "Modbus_Send_Receive".Extrusora_13.Ligado,
                 Heating => "Modbus_Send_Receive".Extrusora_13.Heating,
                 Cooling => "Modbus_Send_Receive".Extrusora_13.Cooling,
                 Fan => "Modbus_Send_Receive".Extrusora_13.Fan,
                 Sts_Fan => "Modbus_Send_Receive".Extrusora_13.Sts_Fan,
                 Sts_Heating => "Modbus_Send_Receive".Extrusora_13.Sts_Heating,
                 Sts_Cooling => "Modbus_Send_Receive".Extrusora_13.Sts_Cooling,
                 Slave => "Modbus_Send_Receive".Extrusora_13.Slave,
                 Master => "Modbus_Send_Receive".Extrusora_13.Master,
                 SP_Out => "Modbus_Send_Receive".Extrusora_13.SP,
                 PV_Out => "Modbus_Send_Receive".Extrusora_13.PV,
                 Malfunction => "Modbus_Send_Receive".Malfunction_13);
END_REGION

REGION Network 14: Extrusora 14
   RUNG wire#powerrail
      "Word_2_Bool"("1_registrador_in" := "Modbus_Send_Receive_1".Reading_Struct."32079", "2_registrador_in" := "Modbus_Send_Receive_1".Reading_Struct."32080", "3_registrador_in" := "Modbus_Send_Receive_1".Reading_Struct."32081", "4_registrador_in" := "Modbus_Send_Receive_1".Reading_Struct."32082", "5_registrador_in" := "Modbus_Send_Receive_1".Reading_Struct."32083", Fancoil_Ligado => "Modbus_Send_Receive".Extrusora_14.Ligado, Heating => "Modbus_Send_Receive".Extrusora_14.Heating, Cooling => "Modbus_Send_Receive".Extrusora_14.Cooling, Fan => "Modbus_Send_Receive".Extrusora_14.Fan, Sts_Fan => "Modbus_Send_Receive".Extrusora_14.Sts_Fan, Sts_Heating => "Modbus_Send_Receive".Extrusora_14.Sts_Heating, Sts_Cooling => "Modbus_Send_Receive".Extrusora_14.Sts_Cooling, Slave => "Modbus_Send_Receive".Extrusora_14.Slave, Master => "Modbus_Send_Receive".Extrusora_14.Master, SP_Out => "Modbus_Send_Receive".Extrusora_14.SP, PV_Out => "Modbus_Send_Receive".Extrusora_14.PV, Malfunction => "Modbus_Send_Receive".Malfunction_14)
   END_RUNG
   // the same network as SCL:
   "Word_2_Bool"("1_registrador_in" := "Modbus_Send_Receive_1".Reading_Struct."32079",
                 "2_registrador_in" := "Modbus_Send_Receive_1".Reading_Struct."32080",
                 "3_registrador_in" := "Modbus_Send_Receive_1".Reading_Struct."32081",
                 "4_registrador_in" := "Modbus_Send_Receive_1".Reading_Struct."32082",
                 "5_registrador_in" := "Modbus_Send_Receive_1".Reading_Struct."32083",
                 Fancoil_Ligado => "Modbus_Send_Receive".Extrusora_14.Ligado,
                 Heating => "Modbus_Send_Receive".Extrusora_14.Heating,
                 Cooling => "Modbus_Send_Receive".Extrusora_14.Cooling,
                 Fan => "Modbus_Send_Receive".Extrusora_14.Fan,
                 Sts_Fan => "Modbus_Send_Receive".Extrusora_14.Sts_Fan,
                 Sts_Heating => "Modbus_Send_Receive".Extrusora_14.Sts_Heating,
                 Sts_Cooling => "Modbus_Send_Receive".Extrusora_14.Sts_Cooling,
                 Slave => "Modbus_Send_Receive".Extrusora_14.Slave,
                 Master => "Modbus_Send_Receive".Extrusora_14.Master,
                 SP_Out => "Modbus_Send_Receive".Extrusora_14.SP,
                 PV_Out => "Modbus_Send_Receive".Extrusora_14.PV,
                 Malfunction => "Modbus_Send_Receive".Malfunction_14);
END_REGION
END_FUNCTION
